// TIA Portal V18 export
TYPE "PresetType"
END_TYPE
